FUNCTION_BLOCK FB_BaseHMIGroupElement_Command EXTENDS FB_BaseHMIControlElement_Command IMPLEMENTS ITF_BaseHMIGroupElement_Command
VAR
END_VAR

END_FUNCTION_BLOCK

(* stored: Version 1.1.0.1
   POU FB_BaseHMIGroupElement_Command: Id {e5955491-d1ec-06ed-0a8c-e1f687a1a6b0}, SpecialFunc None *)
